TYPE E_LOG_HandlerName_OLD :
(

		//E_LOG_OKCONECCTIONTOFSS,
		//E_LOG_LOSTCONECCTIONTOFSS,
		//E_LOG_DOOROPENZONE1,
		//E_LOG_DOOROPENZONE2,
		//E_LOG_STARTBUTTONPRESSED,
		//E_LOG_STOPBUTTONPRESSED,
		//E_LOG_RESETBUTTONPRESSED,
		//E_LOG_EUCANOTRUNNINGPT,
		//E_LOG_EUCANOTRUNNINGCT,
		//E_LOG_TPDNOTRUNNINGPT,
		//E_LOG_TPDNOTRUNNINGCT,
		//E_LOG_EXTNOTRUNNINGPT,
		//E_LOG_EXTNOTRUNNINGCT,
		//E_LOG_MACHINESTATEPT,
		//E_LOG_MACHINESTATECT,
		//E_LOG_PA1ADDED,
		//E_LOG_PA2ADDED,
		//E_LOG_PA3ADDED,
		//E_LOG_INTERIMDIAG1,
		//E_LOG_INTERIMDIAG2,
		//E_LOG_INTERIMDIAG3,
		//E_LOG_STACKOUTOFSEQ,
		//E_LOG_OUTERCOMPLETE,
		//E_LOG_LASTOCVCONTENT,
		//E_LOG_LASTPRINTER04COMMAND,
		//E_LOG_LASTPRINTER05COMMAND,
		//E_LOG_LASTOACCONTENT,
		//E_LOG_ROWCOMPLETE,
		//E_LOG_LAYERCOMPLETE,
		//E_LOG_INTERMEDIATECOMPLETE,
		//E_LOG_CASECOMPLETE,
		//E_LOG_CASEDISCHARGERT,
		//E_LOG_CASEDISCHARGEFT,
		//E_LOG_CASELABELVALIDATION,
		//E_LOG_OUTERAGGREGATIONCODE,
		//E_LOG_ROWCOMPLETECODES,
		//E_LOG_LAYERCOMPLETECODES,
		//E_LOG_FINALISECASECONTENTCODES,
		//E_LOG_INTERPUSHOVERWIRTTEN,
		//E_LOG_CASECOMPLETEOVERWITTEN,
		//E_LOG_CASEDISCHARGEOVERWRITTEN,
		//E_LOG_REJECTEDBYCASEPACKER,
		//E_LOG_CASELABELCODE,
		//E_LOG_MCCREATEDEVENT,
		//E_LOG_CASEVALIDATIONRT,
		//E_LOG_CASEVALIDATIONFT,
		//E_LOG_OCVWRITEERROR,
		//E_LOG_OACWRITEERROR,
		//E_LOG_CACWRITEERROR,
		//E_LOG_CHMWRITEERROR,
		//E_LOG_MLFILLINSTATUS,
		//E_LOG_MLSTATUS,
		//E_LOG_MLRESOTRESTATUS,
		//E_LOG_CODEDIAG1,
		//E_LOG_CODEDIAG2,
		//E_LOG_CODEDIAG3,
		//E_LOG_CODEDIAG4,
		//E_LOG_MASTERLISTDOOR,
		//E_LOG_AGGREGATIONDOOR,
		//E_LOG_WRAPPERDOOR,
		//E_LOG_WRAPPERREJECT1
		//E_LOG_WRAPPERREJECT2



);
END_TYPE

(* stored: Version 1.1.0.1
   DUT E_LOG_HandlerName_OLD: Id {6b4fd51a-4c66-4ef8-9cc7-682584800ea1} *)
